{attribute 'enable_dynamic_creation'}
FUNCTION_BLOCK FutureMCMoveRelative EXTENDS FB_AbstructFuture
VAR_INPUT
END_VAR
VAR_OUTPUT
END_VAR
VAR
	_fb_move_rel	: MC_MoveRelative;
	_executor		: FB_Executor;
	_axis: REFERENCE TO AXIS_REF;
	_distance : MC_LREAL;
	_velocity : MC_LREAL;
	_acceleration: MC_LREAL;
	_deceleration: MC_LREAL;
	_jerk		: MC_LREAL;
	_option : ST_MoveOptions;
	_buffer_mode : MC_BufferMode ;
	_error_id :UDINT;
	_exec_state : UDINT;
	_abort_state : UINT;
END_VAR

METHOD abort : BOOL // Return TRUE if finish.
VAR_INST
	future_halt : FutureMcHalt;
END_VAR
CASE _abort_state OF
	0:
		_exec_state := 0;
		future_halt.set_parameters(_axis, _deceleration, _jerk);
		future_halt.future_name := 'HALT MOVE_RELATIVE';
		_executor.future := future_halt;
		_abort_state := 1;
	1:
		IF _executor.execute() AND _executor.nErrorID = 0 THEN
			_abort_state := 2;
		END_IF
		
		IF _executor.current_state = E_FutureExecutionState.wait_for_process THEN
			_executor.start();
		END_IF
	2:
		abort := TRUE;
END_CASE
END_METHOD

METHOD execute : BOOL // Return TRUE if finish.

CASE _exec_state OF
	0:
		_abort_state := 0;
		_fb_move_rel(Axis := _axis,Execute := FALSE);
		_fb_move_rel(
			Execute := TRUE,
			Axis := _axis,
			Distance := _distance,
			Velocity := _velocity,
			Acceleration := _acceleration,
			Deceleration := _deceleration,
			Jerk := _jerk,
			BufferMode := _buffer_mode,
			Options := _option
		);
		_exec_state := 1;
	1:
		IF _fb_move_rel.Busy THEN
			_fb_move_rel(Axis := _axis,Execute := FALSE);
		END_IF
END_CASE

_error_id := _fb_move_rel.ErrorID;
execute := _fb_move_rel.Done OR _fb_move_rel.Error;
END_METHOD

METHOD init : BOOL // Return TRUE if finish.

VAR
	axis: INT;
END_VAR
_exec_state := 0;
_abort_state := 0;
_error_id := _fb_move_rel.ErrorID;
init := TRUE;
END_METHOD

PROPERTY nErrorID : UDINT
GET
nErrorID := _error_id;
END_GET
SET
END_SET
END_PROPERTY

METHOD set_options : BOOL
VAR_INPUT
	option : ST_MoveOptions;
END_VAR
_option := option;
END_METHOD

METHOD set_parameters : BOOL
VAR_INPUT
	axis : REFERENCE TO AXIS_REF;
	distance : MC_LREAL;
	velocity : MC_LREAL;
	acceleration	: MC_LREAL;		// Set deceleration in case let moving axis halt.
	deceleration	: MC_LREAL;		// Set deceleration in case let moving axis halt.
	jerk			: MC_LREAL;		// Set jerk in case let moving axis halt.
	buffer_mode : MC_BufferMode;
END_VAR
_axis REF= axis;
_distance := distance;
_velocity := velocity;
_acceleration := acceleration;
_deceleration := deceleration;
_jerk := jerk;
_buffer_mode := buffer_mode;
END_METHOD

END_FUNCTION_BLOCK

(* stored: Version 1.1.0.1, ProductVersion 3.1.4024.12
   POU FutureMCMoveRelative: Id {68392a9c-c48d-4da1-9d24-d5280f44f2c9}, SpecialFunc None
   Method abort: Id {8d2f52e3-49e4-4662-be7f-97ff2c46b0a5}
   Method execute: Id {20088402-d158-4220-ba48-4075b6c9821d}
   Method init: Id {4a5527fb-69f1-4f27-99bf-902e0f84d9fa}
   Property nErrorID: Id {b27d20ec-8fe1-4336-adde-3ef6b9ae6a52}
   Get Get: Id {1496e878-37c0-4d07-a5bd-a2d02738b4ee}
   Set Set: Id {f5d494bb-e982-49c9-bf0a-301e76f48535}
   Method set_options: Id {026c747f-8220-4684-ae1b-5229a3fc953e}
   Method set_parameters: Id {38aa7173-6e5a-4ac4-8011-d9e2cedddd6f} *)
